(* IEC 61131-3 sources: paho.mqtt.c-ar/Samples/IotMqttSamples/SampleTasks/SSL, 3 files *)

(* ---- Main.st ---- *)
PROGRAM _CYCLIC

	Parameters;

	IotMqttClient_0.Enable			:= TRUE;
	IotMqttClient_0.Connect			:= TRUE;
	IotMqttClient_0.IotMqttLink 	:= ADR(IotMqttLink);
	IotMqttClient_0.Parameters		:= IotMqttParameters;
	IotMqttClient_0();

	PublishTopic	:= 'B&R_DemoProject/SSL';
	brsstrcat(ADR(PublishTopic),ADR(ClientID));

	Subscribe;
	Publish;
END_PROGRAM

PROGRAM _EXIT

    IotMqttClient_0(Enable	:= FALSE);
    IotMqttPublish_0(Enable	:= FALSE);
    IotMqttSubscribe_0(Enable := FALSE);

END_PROGRAM

(* ---- Parameters.st ---- *)
ACTION Parameters:

	//Prepare Client ID. Add a timestamp to ensure any client will repeat it
	UtcDTGetTime_0(enable := TRUE);
	IF brsstrcmp(ADR(ClientID),ADR('')) = 0 THEN
		ClientID := 'B&R_Demo_';
		ST_name(0,ADR(ThreadName),0);
		brsstrcat(ADR(ClientID),ADR(ThreadName));
		brsstrcat(ADR(ClientID),ADR("_"));
		brsmemset(ADR(AuxString),0,SIZEOF(AuxString));
		AuxString := UDINT_TO_STRING(DT_TO_UDINT(UtcDTGetTime_0.DT1));
		brsstrcat(ADR(ClientID),ADR(AuxString));	//Timestamp
	END_IF

	IotMqttParameters.ServerUri				:= 'test.mosquitto.org';
	IotMqttParameters.ConnectionType		:= IotMqtt_TCP;	//Use standard tcp with tls
	IotMqttParameters.Port					:= 8883;
	IotMqttParameters.TLS.UseTLS			:= TRUE;
	IotMqttParameters.ClientID				:= ClientID;
	IotMqttParameters.CleanSession			:= TRUE;
	IotMqttParameters.KeepAliveInterval		:= T#20s;
	IotMqttParameters.AutomaticReconnect	:= TRUE;

END_ACTION

(* ---- Publish.st ---- *)
ACTION Publish:

	IF CmdAutoPublish THEN
		IF (IotMqttPublish_0.Done OR IotMqttPublish_0.Error) AND IotMqttClient_0.Connected THEN
			IotMqttPublish_0.Send := FALSE;
		ELSIF IotMqttClient_0.Connected THEN
			IotMqttPublish_0.Send := TRUE;
		END_IF;
	END_IF

	brsmemset(ADR(PublishMessage),0,SIZEOF(PublishMessage));
	brsmemset(ADR(AuxString),0,SIZEOF(AuxString));
	PublishMessage := ClientID;
	brsstrcat(ADR(PublishMessage),ADR(' Test message #'));
	AuxString := UDINT_TO_STRING(IotMqttPublish_0.Info.MessagesPublished);
	brsstrcat(ADR(PublishMessage),ADR(AuxString));

	IotMqttPublish_0.Enable			:= TRUE;
	IotMqttPublish_0.IotMqttLink	:= IotMqttClient_0.IotMqttLink;
	IotMqttPublish_0.Topic			:= ADR(PublishTopic);
	IotMqttPublish_0.QoS			:= IotMqtt_QoS0;
	IotMqttPublish_0.Buffer			:= ADR(PublishMessage);
	IotMqttPublish_0.BufferLength	:= brsstrlen(ADR(PublishMessage));
	IotMqttPublish_0.Retained		:= FALSE;

	IotMqttPublish_0();

END_ACTION
